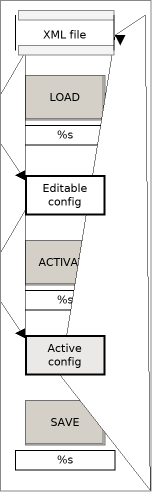
VISUALIZATION VISU_ConfigManager  // 152x492
VAR_IN_OUT
	mgr : ConfigManager;
    widget : ConfigManagerWidget;
END_VAR
    Button (25,75 80x45), "LOAD", input disabled if: mgr.processes.load.statuses.enabledStatus.disabled
        OnMouseClick: execute { mgr.processes.load.do_request := TRUE; }
    Button (25,240 80x45), "ACTIVATE", input disabled if: mgr.processes.activate.statuses.enabledStatus.disabled
        OnMouseClick: execute { mgr.processes.activate.do_request := TRUE; }
    Rectangle (15,125 100x20), "%s", text variable: widget.load.description, colour variable: widget.load.bgColor
        p55702900: widget.load.fgColor
    Rectangle (15,290 100x20), "%s", text variable: widget.load.description, colour variable: widget.load.bgColor
        p55702900: widget.load.fgColor
    Button (25,400 80x45), "SAVE", input disabled if: mgr.processes.save.statuses.enabledStatus.disabled
        OnMouseClick: execute { mgr.processes.save.do_request := TRUE; }
    Rectangle (15,450 100x20), "%s", text variable: widget.save.description, colour variable: widget.save.bgColor
        p55702900: widget.load.fgColor
    Polygon (25,52) (0,95) (-5,135) (25,180)
    Polygon (15,175) (25,170) (25,180)
    Polygon (25,210) (0,253) (-5,293) (25,338)
    Polygon (15,333) (25,328) (25,338)
    Polygon (60,375) (150,490) (145,15) (115,35)
    Polygon (115,35) (125,35) (120,45)
    RoundedRectangle (25,175 80x40), "Editable config"
    Pie (18,45 96x10)
    Pie (18,10 96x10)
    Line (114,50) (114,15)
    RoundedRectangle (25,335 80x40), "Active config"
    Label (20,20 90x30), "XML file"
    Line (15,15) (15,50)
END_VISUALIZATION

(* stored: Version 1.1.0.1, ProductVersion 3.1.4019.2
   Visu VISU_ConfigManager: Id {6b29a266-f5d8-4639-9b47-3367ab10f2a7} *)
